TYPE udt_HDL_PartData :
STRUCT
	
PartId	:DINT;
State	:BOOL;
Varient	:BOOL;
Exists	:BOOL;

	
END_STRUCT
END_TYPE

(* stored: Version 1.1.0.1, ProductVersion 3.1.4024.16
   DUT udt_HDL_PartData: Id {bc52548c-555b-48bb-95ee-c28b2ac877ed} *)
